// TIA Portal V17 export
// export: Created 2024-06-14T09:53:47.0057171Z, ExportSetting WithDefaults, DisplayName Totally Integrated Automation Portal, DisplayVersion V17, DisplayName TIA Portal Openness, DisplayVersion V17, DisplayName TIA Portal Version Control Interface, DisplayVersion V17, DisplayName Simotion SCOUT TIA, DisplayVersion 5.4.3.0, DisplayName SINAMICS Startdrive Advanced, DisplayVersion V17 SP1 Update 1, DisplayName SINAMICS Startdrive G110M, G120, G120C, G120D, G120P, G115D, DisplayVersion V17 SP1 Update 1, DisplayName SINAMICS Startdrive G130, G150, S120, S150, SINAMICS MV, S210, DisplayVersion V17 SP1 Update 1, DisplayName STEP 7 Professional, DisplayVersion V17, DisplayName STEP 7 Safety, DisplayVersion V17, DisplayName WinCC Professional, DisplayVersion V17
VAR_GLOBAL   // PLC tag table "Fine Filling Station-4"
   S4_CYCLE_START AT %I0.0 : Bool;
   S4_CYCLE_RESET AT %I0.1 : Bool;
   S4_STOPPER_SENSOR AT %I2.3 : Bool;
   S4_SENSOR_CYL1 AT %I1.1 : Bool;
   S4_SENSOR_CYL2 AT %I1.2 : Bool;
   S4_SENSOR_CYL3 AT %I1.3 : Bool;
   S4_SENSOR_CYL4 AT %I1.4 : Bool;
   S4_SENSOR_CYL5 AT %I1.5 : Bool;
   S4_SENSOR_CYL6 AT %I1.6 : Bool;
   SPARE_1 AT %I1.7 : Bool;
   MANUAL_SEQ_L2 AT %I2.0 : Bool;
   "i0.6_L2" AT %I2.1 : Bool;
   "i0.7_L2" AT %I2.2 : Bool;
   S4_DOWN_CONVEYOR AT %I1.0 : Bool;
   S4_STOPPER_OP AT %Q0.1 : Bool;
   S4_LIFT_CYL1 AT %Q0.2 : Bool;
   S4_LIFT_CYL2 AT %Q0.3 : Bool;
   S4_LIFT_CYL3 AT %Q0.4 : Bool;
   S4_LIFT_CYL4 AT %Q0.5 : Bool;
   S4_LIFT_CYL5 AT %Q0.6 : Bool;
   S4_LIFT_CYL6 AT %Q0.7 : Bool;
   S4_LIFT_CYL7 AT %Q1.0 : Bool;
   S4_LIFT_CYL8 AT %Q1.1 : Bool;
   S4_LIFT_CYL9 AT %Q1.2 : Bool;
   S4_LIFT_CYL10 AT %Q1.3 : Bool;
   S5_LIFT_CYL4 AT %Q2.3 : Bool;
   S5_LIFT_CYL3 AT %Q2.4 : Bool;
   S5_LIFT_CYL2 AT %Q2.5 : Bool;
   S5_LIFT_CYL1 AT %Q2.6 : Bool;
   spare_11 AT %Q2.7 : Bool;
   spare_12 AT %Q3.0 : Bool;
   spare_13 AT %Q3.1 : Bool;
   spare_14 AT %Q3.2 : Bool;
   spare_15 AT %Q3.3 : Bool;
   spare_16 AT %Q3.4 : Bool;
END_VAR
